(* CoDeSys 2.3 export: STRPUMPCONTROLBUTTON.EXP *)

(* Data type *)
TYPE strPumpControlButton :
STRUCT
	on : BOOL;
	off: BOOL;
END_STRUCT
END_TYPE
